PROGRAM PRG_Test
VAR
	anyTypeBindedTest : AnyTypeTest;
	boolBindingReadOnlyTest : BoolBindingReadOnlyTest;
	bindTest : BindTest;
	notBindTest : NotBindTest;
	
	reflectionTest : ReflectionTest;
	
	boolValuesTest : BoolValuesTest;
	booleanExpressionTest : BooleanExpressionTest;
	booleanExpressionFunctionsTest : BooleanExpressionFunctionsTest;
END_VAR

TcUnit.RUN();

END_PROGRAM

(* stored: Version 1.1.0.1, ProductVersion 3.1.4024.12
   POU PRG_Test: Id {59fba049-dffd-419e-9eb9-7a7800aaf4f4}, SpecialFunc None *)
